PROGRAM MAIN
VAR
	fbAmericanSalamiPizza		: FB_Pizza(ePizzaStyle := E_PizzaStyle.eAmerican, bHasBroccoli := FALSE, bHasCheese := TRUE, bHasSalami := TRUE);
	fbItalianVegetarianPizza	: FB_Pizza(ePizzaStyle := E_PizzaStyle.eItalian, bHasBroccoli := TRUE, bHasCheese := FALSE, bHasSalami := FALSE);
END_VAR

END_PROGRAM

(* stored: Version 1.1.0.1, ProductVersion 3.1.4022.12
   POU MAIN: Id {8628af66-e1f3-48a0-aced-3f5f2bc2e309}, SpecialFunc None *)
